PROGRAM BkgrdSerialLaser
VAR
	(* background communication with the EL6002 terminal *)
	serialLineCtrl		: SerialLineControl;
	serialLineCtrlError	: BOOL;
	serialLineCtrlErrorID : ComError_t;
	(* 	I/O variables for a EL6002 terminal*)
	stInLaser  AT %I* : EL6inData22B;	
	stOutLaser AT %Q* : EL6outData22B;
END_VAR

(*
The SerialLineControl function block is supposed to be called in every PLC cycle.
It communicates with the serial line hardware device and transmits or receives data.
The SerialLineControl can be called in the standard task (e.g.for PcCOM port usage) 
or in a separate fast task (e.g.for terminal usage) as well.
A fast separate task will be necessary at high baud rates or with KL6001 terminals 
which have a small process image (3 or 5 data bytes only)
*)

(* background communication with the EL6002 terminal *)
serialLineCtrl(
	Mode:= SERIALLINEMODE_EL6_22B, 
	pComIn:= ADR(stInLaser), 
	pComOut:= ADR(stOutLaser), 
	SizeComIn:= SIZEOF(stInLaser), 
	TxBuffer:= HardwareGlobalVariables.TxBufferLaser, 
	RxBuffer:= HardwareGlobalVariables.RxBufferLaser
);

IF serialLineCtrl.Error THEN
	serialLineCtrlError := TRUE;
	serialLineCtrlErrorID := serialLineCtrl.ErrorID;
END_IF

END_PROGRAM

(* stored: Version 1.1.0.1, ProductVersion 3.1.4024.4
   POU BkgrdSerialLaser: Id {878cee48-a19e-46ed-8231-c216b4e804ac}, SpecialFunc None *)
